FUNCTION_BLOCK AX_TOF (* Standard timer function block (off-delay timing) *)
  (* Standard: 61499-2; Classification: standard timer function block; Description: Copyright (c) 2024 HR Agrartechnik GmbH This program and the accompanying materials are made available under the terms of the Eclipse Public License 2.0 which is available at https://www.eclipse.org/legal/epl-2.0/ SPDX-License-Identifier: EPL-2.0 AX_TOF -- Off-delay timer FB with AX adapter interface The adapter input IN triggers execution (E1->REQ) and provides the boolean input value (D1->IN). The event input R presets the off-delay time PT and resets the timer. When IN goes TRUE, Q becomes TRUE immediately. When IN goes FALSE, Q stays TRUE for duration PT before going FALSE. Reset stops the timer and sets Q to FALSE. *)
  (* Version 3.0, 2025-04-14, Patrick Aigner, changed package *)
  (* Version 1.1, 2024-04-23, Franz Höpfinger, HR Agrartechnik GmbH, Add a Reset to Timer FBs *)
  (* Version 1.0, 2024-03-04, Franz Höpfinger, HR Agrartechnik GmbH *)
  PACKAGE adapter::events::unidirectional::timers;
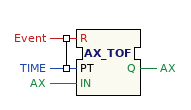
  EVENT_INPUT
    R WITH PT; (* Reset *)
  END_EVENT
  VAR_INPUT
    PT : TIME; (* Off-delay time *)
  END_VAR
  SOCKETS
    IN : adapter::types::unidirectional::AX; (* Timer input (AX adapter) *)
  END_SOCKETS
  PLUGS
    Q : adapter::types::unidirectional::AX; (* Timer output (AX adapter) *)
  END_PLUGS
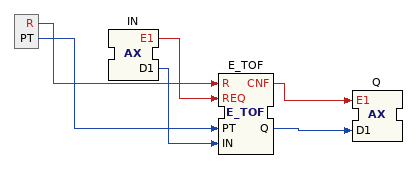
  FBS
    E_TOF : iec61499::events::timers::E_TOF;
  END_FBS
  EVENT_CONNECTIONS
    R TO E_TOF.R;
    E_TOF.CNF TO Q.E1;
    IN.E1 TO E_TOF.REQ;
  END_CONNECTIONS
  DATA_CONNECTIONS
    PT TO E_TOF.PT;
    E_TOF.Q TO Q.D1;
    IN.D1 TO E_TOF.IN;
  END_CONNECTIONS
END_FUNCTION_BLOCK
